FUNCTION_BLOCK Q_BackgroundColour (* Command change background colour ( Part 6 - F.20 ) *)
  (* Standard: ISO 11783-6; Description: This command is used to change the background colour of an object. etval iso_s16 - #E_NO_ERR - OK - #E_OVERFLOW - buffer overflow - #E_NOACT - Command not possible in current state - #E_NO_INSTANCE - No VT client available *)
  (* Version 1.0, 2022-07-08, franz *)
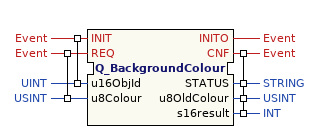
  EVENT_INPUT
    INIT WITH u16ObjId; (* Service Initialization *)
    REQ WITH u8Colour; (* Service Request *)
  END_EVENT
  EVENT_OUTPUT
    INITO; (* Initialization Confirm *)
    CNF WITH STATUS, u8OldColour, s16result; (* Confirmation of Requested Service *)
  END_EVENT
  VAR_INPUT
    u16ObjId : UINT; (* Object ID *)
    u8Colour : USINT; (* New Background colour see Part 6 - A.3 VT standard colour palette *)
  END_VAR
  VAR_OUTPUT
    STATUS : STRING; (* Service Status *)
    u8OldColour : USINT; (* Old value of ID *)
    s16result : INT; (* retval see description *)
  END_VAR
END_FUNCTION_BLOCK
